(* PLC project  *)

CONFIGURATION CANbus
END_CONFIGURATION
